PROGRAM Stn054_51_Stn321MainMergePrestop
VAR
//correct
	{attribute 'TcLinkToOSO' := '
			.iPuckPresent :=  <0,1,2>TIIB[N58S00 (AL1332)]^N58S01 (AL2341)^TxPDO^input byte 0;
			.iBufferFull  :=  <0,1,2>TIIB[N58S00 (AL1332)]^N58S01 (AL2341)^TxPDO^input byte 2;
			.oStopLower  :=  <0,1,1>TIIB[N58S00 (AL1332)]^N58S02 (EX260)^RxPDO^output byte 0'}
	fbConvStop: FB_ConvStop;
END_VAR

//  This code instantiates a component that is implimented as a common function block
//    Note that I/O is linked directly to I/O variables inside the named instance
//Stn 321 GRN Exit Main Stop Puck Present
//Stn 321 GRN  Exit Main Stop DS Buffer
//Stn321MergeMainPrestop  (1B)

gStn054_51_Stn321MainMergePrestop.ConvRunning  := gConsumed_SafetyInterfaceConv.MtrRunning.Enc058Mtr05 AND gConsumed_SafetyInterfaceConv.MtrRunning.Enc059Mtr01;

fbConvStop(
	pStn := ADR(gStn054),
	pCmp := ADR(gStn054_51_Stn321MainMergePrestop),
	pUpstreamStop := 0,
	pStateTraceBuffer := ADR(gStn054_StateTraceBuffer),
	pStateTraceFifo := ADR(gStn054_StateTraceFifo),
	pStats := ADR(gStn054_02_Stats));

END_PROGRAM

(* stored: Version 1.1.0.1, ProductVersion 3.1.4024.6
   POU Stn054_51_Stn321MainMergePrestop: Id {0928ab4e-e8f9-4e41-9743-b6f6ba022729}, SpecialFunc None *)
